% RSLogix 500 project DIGITAL HEATER CONTROL_BAK000.RSS, saved by version 8.30.00.16 %
PROJECT "UNTITLED"    % processor: Bul.1763 MicroLogix 1100 Series B %

PROGRAM FILES
  LAD 2   10 rungs

DATA FILES
  O0 OUTPUT  9 elements
  I1 INPUT  16 elements
  S2 STATUS  66 elements
  B3 BINARY  1 elements
  T4 TIMER  1 elements
  C5 COUNTER  1 elements
  R6 CONTROL  1 elements
  N7 INTEGER  1 elements
  F8 FLOAT  1 elements

LADDER 2
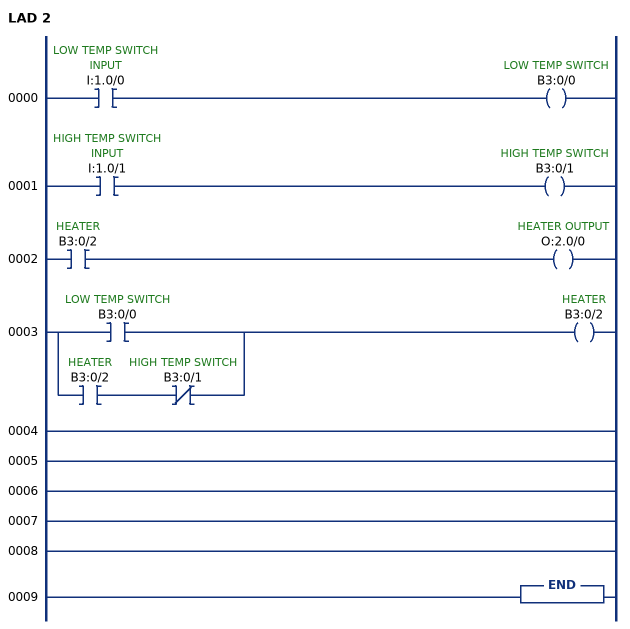
% Rung: 0 %  % edit flag set %
SOR XIC I:1.0/0 OTE B3:0/0 EOR
%   I:1.0/0  "LOW TEMP SWITCH INPUT" %
%   B3:0/0  "LOW TEMP SWITCH" %
% Rung: 1 %  % edit flag set %
SOR XIC I:1.0/1 OTE B3:0/1 EOR
%   I:1.0/1  "HIGH TEMP SWITCH INPUT" %
%   B3:0/1  "HIGH TEMP SWITCH" %
% Rung: 2 %  % edit flag set %
SOR XIC B3:0/2 OTE O:2.0/0 EOR
%   B3:0/2  "HEATER" %
%   O:2.0/0  "HEATER OUTPUT" %
% Rung: 3 %  % edit flag set %
SOR BST XIC B3:0/0 NXB XIC B3:0/2 XIO B3:0/1 BND OTE B3:0/2 EOR
%   B3:0/0  "LOW TEMP SWITCH" %
%   B3:0/2  "HEATER" %
%   B3:0/1  "HIGH TEMP SWITCH" %
% Rung: 4 %  % edit flag set %
SOR EOR
% Rung: 5 %  % edit flag set %
SOR EOR
% Rung: 6 %  % edit flag set %
SOR EOR
% Rung: 7 %  % edit flag set %
SOR EOR
% Rung: 8 %  % edit flag set %
SOR EOR
% Rung: 9 %
SOR END EOR

OTHER DOCUMENTED ADDRESSES
  B3:0/12  "HIGH TEMP SWITCH"
